// TIA Portal V16 export
// export: Created 2024-05-10T06:46:43.3049083Z, ExportSetting WithDefaults, DisplayName Totally Integrated Automation Portal, DisplayVersion V16, DisplayName TIA Portal Version Control Interface, DisplayVersion V16, DisplayName TIA Portal Openness, DisplayVersion V16, DisplayName STEP 7 Professional, DisplayVersion V16, DisplayName STEP 7 Safety, DisplayVersion V16, DisplayName WinCC Professional, DisplayVersion V16
DATA_BLOCK "K04_报警_DB"   // DB4
VERSION : 0.1
// stored: AutoNumber true, DBAccessibleFromOPCUA true, InstanceOfName K04_报警, InstanceOfType FB
"K04_报警"
   // VAR
   //    MT_ErrTime : Array[1..3] of IEC_TIMER;
   // END_VAR
BEGIN
END_DATA_BLOCK
